PROGRAM MAIN
VAR
	xCall				:BOOL;
	AddParams			:M_ADD_Parameters := (A := 40, B := 2);
	MeaningOfLife		:LREAL;
	
	fbRPC				:FB_InvokeRpcMethod;
	xBusy				:BOOL;
	xError				:BOOL;	
	nErrorID			:UDINT;	
END_VAR

fbRPC(
	bCall					:=xCall , 
	sNetId					:='' , 
	nPort					:=851 , 
	sMethodName				:='MAIN.fbMath#M_ADD' , 
	nSrcAddrParameter		:=ADR(AddParams) , 
	nLenParameter			:=SIZEOF(AddParams) , 
	nDestAddrReturnValue	:=ADR(MeaningOfLife) , 
	nLenReturnValue			:=SIZEOF(MeaningOfLife) , 
	tTimeout				:=DEFAULT_ADS_TIMEOUT , 
	eComMode				:=E_AdsComMode.eAdsComModeFastCom , 
	bBusy					=>xBusy , 
	bError					=>xError , 
	nErrorId				=>nErrorID );

END_PROGRAM

(* stored: Version 1.1.0.1, ProductVersion 3.1.4024.11
   POU MAIN: Id {e4d3bc24-10d3-4594-9f36-0dd39168eed0}, SpecialFunc None *)
